{attribute 'qualified_only'}
{attribute 'strict'}
TYPE SetPointTypes :
(
	Standard := 0, Alternative
);
END_TYPE

(* stored: Version 1.1.0.1, ProductVersion 3.1.4024.6
   DUT SetPointTypes: Id {73abc6dc-1bf0-4b66-ad19-b8082a03c809} *)
